(* CODESYS project codesys-demo

Project tree, tasks and I/O mapping:
  Device : CODESYS Control Win V3, 3S - Smart Software Solutions GmbH, version 3.5.17.0
    application Application
      libraries: Standard, * (System)
      task MainTask (cyclic, interval t#20ms, priority 1) calls PLC_PRG
      program PLC_PRG [ST]
*)

// Device/Application/PLC_PRG
PROGRAM PLC_PRG
VAR
END_VAR

END_PROGRAM
